INTERFACE I_HController

END_INTERFACE

(* stored: Version 1.1.0.1
   Itf I_HController: Id {c93b96fa-8d4c-48a2-b6f1-b4ec09d8c803} *)
